FUNCTION_BLOCK KukaRobot
VAR_OUTPUT
	(*
	forceStop AT %Q* : BOOL;
	resetSignal AT %Q* : BOOL;
	*)
	
	reservation : INT := 0;
	
	error : BOOL;
	errorID : DINT;
	
	outputs AT %Q* : ARRAY[1..20] OF WORD;
	inputs AT %I* : ARRAY[1..20] OF WORD;
END_VAR
VAR
	heartbeat : Watchdog;
	
	offline AT %I* : BOOL;
	toggleBit AT %I* : BOOL;
	
	hmiReservation : STRING;
END_VAR
(*
generic KUKA robot with 20 WORD outputs and 20 WORD inputs, connected to Beckhoff IPC via EL6692 or EL6695 EtherCAT bridge
includes minimal diagnostics to detect if robot is offline
robots should always be reserved before sending a task
*)

heartbeat(
	enable:= NOT offline,
	toggleBit:= toggleBit,
	timeoutWidth:= T#200MS,
	timeout=> );

error := //add any addition conditions with OR
	offline OR
	heartbeat.timeout;

//{attribute 'monitoring' := 'variable'}
{attribute 'monitoring' := 'call'}
PROPERTY Busy : BOOL
GET
END_GET
END_PROPERTY

METHOD clearCommand : BOOL
VAR_INPUT
	reserveID : INT;
END_VAR
IF reservation = reserveID THEN
	MEMSET(ADR(outputs), 0, SIZEOF(outputs));
END_IF
END_METHOD

//{attribute 'monitoring' := 'variable'}
{attribute 'monitoring' := 'call'}
PROPERTY Done : BOOL
GET
END_GET
END_PROPERTY

{attribute 'monitoring' := 'call'}
PROPERTY Ready : BOOL
GET
END_GET
END_PROPERTY

METHOD release : BOOL
VAR_INPUT
	reserveID : SectionEnum;
END_VAR
IF reservation = reserveID THEN
	reservation := SectionEnum.NULL_SECTION;
	release := TRUE;
END_IF
END_METHOD

METHOD reserve : BOOL
VAR_INPUT
	reserveID : INT;
END_VAR
(*
this method exists because chipboard and wood bunk operations use the same robot
both sections need to check if the robot is open to commands before use
*)
IF Reserved AND reservation = reserveID THEN
	reserve := TRUE;

ELSIF NOT Reserved THEN
	reservation := reserveID;
	reserve := TRUE;

END_IF
END_METHOD

{attribute 'monitoring' := 'call'}
PROPERTY Reserved : BOOL
GET
Reserved := reservation <> SectionEnum.NULL_SECTION;
END_GET
END_PROPERTY

METHOD reset : BOOL
//resetSignal := TRUE;
//done := FALSE;

MEMSET(ADR(outputs), 0, SIZEOF(outputs));
(*
IF ready AND completedTask = 0 THEN
	resetSignal := FALSE;
	reset := TRUE;
END_IF
*)
END_METHOD

METHOD resume : BOOL
//forceStop := FALSE;

resume := NOT error AND errorID = 0;
END_METHOD

METHOD setGroup : BOOL
VAR_INPUT
	reserveID : INT;
	group : INT;
	value : INT;
END_VAR
{warning disable C0195}
IF reservation = reserveID THEN
	outputs[group] := value;
	setGroup := TRUE;
END_IF
END_METHOD

METHOD stop : BOOL
VAR_INPUT
END_VAR
//forceStop := TRUE;
stop := TRUE;

//MEMSET(ADR(outputs), 0, SIZEOF(outputs));
END_METHOD

END_FUNCTION_BLOCK

(* stored: Version 1.1.0.1, ProductVersion 3.1.4024.11
   POU KukaRobot: Id {60b8c04d-38ba-483d-baa2-feca47e063a5}, SpecialFunc None
   Folder Properties: Id {8ffe1e39-61c1-4398-8ddf-38564de07f51}
   Property Busy: Id {152763dc-c4e3-4017-bc80-d712b47856e1}
   Get Get: Id {7a14ab38-ad73-468e-a307-13933f79a0c1}
   Method clearCommand: Id {24ee99e9-db60-47bb-8bfa-bceffbdd3e3c}
   Property Done: Id {08daa405-24a1-4c74-b41d-88b33003f753}
   Get Get: Id {4d1fb0e6-4d99-44c5-bc16-89b50d9e21bd}
   Property Ready: Id {9650ecd7-d852-4b27-ba50-624c1407563d}
   Get Get: Id {efd257b8-0901-4188-afa5-ec7a19fa1b9e}
   Method release: Id {9cb9c870-9a0a-4e25-9e69-66c536dd5de8}
   Method reserve: Id {105269a9-e981-4b0d-a0fb-dab94fd22a02}
   Property Reserved: Id {e6648a14-0c6c-4acd-ab38-8227ede6160b}
   Get Get: Id {9ba9db71-1fc5-478e-9511-6f7e0a894756}
   Method reset: Id {e89fe8c1-79a5-4653-863f-2064d194b5df}
   Method resume: Id {6e4c2487-3770-49c6-bd78-e95a5e370aa9}
   Method setGroup: Id {1af94f2c-ccd7-455d-a302-323d49e91687}
   Method stop: Id {9d09e203-8c3b-40f7-893c-e33c2349a4ff} *)
